// TwinCAT 3 PLC project mobject_nci
// Title: mobject-nci
// Company: mobject-io-ext
// Author: mobject dev team
// ProjectVersion: 0.0.1
// ProgramVersion: 3.1.4023.0
// libraries:
//   mobject-core, * (mobject.io)
//   mobject-motion, * (mobject-io-ext)
//   Tc2_NCI, * (Beckhoff Automation GmbH)
//   Tc2_PlcInterpolation, * (Beckhoff Automation GmbH)
//   Tc3_Module, * (Beckhoff Automation GmbH)
// project tree:
//   Lib/Feeder/ Feeder.TcPOU, I_Feeder.TcIO
//   Lib/NC-I/ ChannelType.TcDUT, I_Nci.TcIO, Nci.TcPOU, NciAxis.TcDUT, NciPlc.TcDUT
//   Lib/NC-I/Commands/ AddAxisToGroupCommand.TcPOU, BuildXYZGroupCommand.TcPOU, I_NciCommand.TcIO, NciCommand.TcPOU, ReleaseAxisCommand.TcPOU, ResetGroupCommand.TcPOU
//   Lib/Table/Enums/ FeedrateInterpolation.TcDUT, StandardPlane.TcDUT, TangentialFollowingBehaviour.TcDUT, VertexSmoothingBlendingType.TcDUT, VertexSmoothingSubType.TcDUT
//   Lib/Table/ I_Table.TcIO, Table.TcPOU

// ---- Lib/NC-I/ChannelType.TcDUT
{attribute 'qualified_only'}
{attribute 'strict'}
TYPE ChannelType :
(
	NONE := Tc2_PlcInterpolation.E_ItpChannelType.ItpChannelTypeNone,
	INTERPRETER := Tc2_PlcInterpolation.E_ItpChannelType.ItpChannelTypeInterpreter,
	KINEMATIC := Tc2_PlcInterpolation.E_ItpChannelType.ItpChannelTypeKinematic,
	INVALID_ITF_VERSION := Tc2_PlcInterpolation.E_ItpChannelType.ItpChannelType_InvalidItfVer
) INT;
END_TYPE

// ---- Lib/NC-I/NciAxis.TcDUT
{attribute 'qualified_only'}
{attribute 'strict'}
TYPE NciAxis :
(
	NONE := Tc2_PlcInterpolation.E_NciAxesInGroup.NoneAxis,
	X_AXIS := Tc2_PlcInterpolation.E_NciAxesInGroup.XAxis,
	Y_AXIS := Tc2_PlcInterpolation.E_NciAxesInGroup.YAxis,
	Z_AXIS := Tc2_PlcInterpolation.E_NciAxesInGroup.ZAxis,
	Q1_AXIS := Tc2_PlcInterpolation.E_NciAxesInGroup.Q1Axis,
	Q2_AXIS := Tc2_PlcInterpolation.E_NciAxesInGroup.Q2Axis,
	Q3_AXIS := Tc2_PlcInterpolation.E_NciAxesInGroup.Q3Axis,
	Q4_AXIS := Tc2_PlcInterpolation.E_NciAxesInGroup.Q4Axis,
	Q5_AXIS := Tc2_PlcInterpolation.E_NciAxesInGroup.Q5Axis
) INT;
END_TYPE

// ---- Lib/NC-I/NciPlc.TcDUT
TYPE NciPlc :
STRUCT
	nciToPlc AT %I* : NcToPlc_NciChannel_Ref;
	plcToNci AT %Q* : PlcToNc_NciChannel_Ref;
END_STRUCT
END_TYPE

// ---- Lib/Table/Enums/FeedrateInterpolation.TcDUT
{attribute 'qualified_only'}
{attribute 'strict'}
TYPE FeedrateInterpolation :
(
	CONST := Tc2_PlcInterpolation.E_NciFeedRateIpol.E_NciFeedrateIpolConstant,
    LINEAR := Tc2_PlcInterpolation.E_NciFeedRateIpol.E_NciFeedrateIpolLinear
) UINT;
END_TYPE

// ---- Lib/Table/Enums/StandardPlane.TcDUT
{attribute 'qualified_only'}
{attribute 'strict'}
TYPE StandardPlane :
(
	XY := Tc2_PlcInterpolation.E_NciGeoPlane.E_NciGeoPlaneXY,
	ZX := Tc2_PlcInterpolation.E_NciGeoPlane.E_NciGeoPlaneZX,
	YZ := Tc2_PlcInterpolation.E_NciGeoPlane.E_NciGeoPlaneYZ
) INT;
END_TYPE

// ---- Lib/Table/Enums/TangentialFollowingBehaviour.TcDUT
{attribute 'qualified_only'}
{attribute 'strict'}
TYPE TangentialFollowingBehaviour :
(
	IGNORE_ALL := Tc2_PlcInterpolation.E_TangentialFollowingBehavior.E_TfIngoreAll, // ignore critical angle
	ERROR_ON_EXCEEDING_CRITICAL_ANGLE := Tc2_PlcInterpolation.E_TangentialFollowingBehavior.E_TfErrorOnCritical1 // if angle becomes bigger than critical angle 1 ==> error
) INT;
END_TYPE

// ---- Lib/Table/Enums/VertexSmoothingBlendingType.TcDUT
{attribute 'qualified_only'}
{attribute 'strict'}
TYPE VertexSmoothingBlendingType :
(
	NONE := 0, // Probably should check this is correct!
	PARABOLIC := 2,
	BI_QUADRATIC := 3,
	BEZIER_3RD_ORDER := 4,
	BEZIER_5TH_ORDER := 5
) UDINT;
END_TYPE

// ---- Lib/Table/Enums/VertexSmoothingSubType.TcDUT
{attribute 'qualified_only'}
{attribute 'strict'}
TYPE VertexSmoothingSubType :
(
	NONE := 0, // Probably should check this is correct!
	CONSTANT_TOLERANCE_RADIUS := 1,
	DISTANCE_BETWEEN_INTERSETION_AND_VERTEX := 2,
	ADAPTIVE_TOLERANCE_RADIUS := 3
) UDINT;
END_TYPE

// ---- Lib/Feeder/I_Feeder.TcIO
INTERFACE I_Feeder EXTENDS __System.IQueryInterface

PROPERTY ChannelDone : BOOL
GET
END_GET
END_PROPERTY

METHOD FeedTable
VAR_INPUT
	table : I_Table;
	feedback : REFERENCE TO I_CommandFeedback;
END_VAR
END_METHOD

PROPERTY LogFeederEntries : BOOL
GET
END_GET
SET
END_SET
END_PROPERTY

METHOD Reset
VAR_INPUT
	feedback : REFERENCE TO I_CommandFeedback;
END_VAR
END_METHOD

END_INTERFACE

// ---- Lib/NC-I/Commands/I_NciCommand.TcIO
INTERFACE I_NciCommand EXTENDS I_Command

END_INTERFACE

// ---- Lib/NC-I/I_Nci.TcIO
INTERFACE I_Nci EXTENDS __System.IQueryInterface

PROPERTY _InternalNciPlcRef : REFERENCE TO NciPlc
GET
END_GET
END_PROPERTY

METHOD AddAxisToGroup
VAR_INPUT
	axis : I_Axis;
	index : UDINT;
	timeout : TIME;
	feedback : REFERENCE TO I_CommandFeedback;
END_VAR
END_METHOD

PROPERTY BlockNumber : UDINT
GET
END_GET
END_PROPERTY

METHOD BuildXYGroup
VAR_INPUT
	xAxis : I_Axis;
	yAxis : I_Axis;
	timeout : TIME;
	feedback : REFERENCE TO I_CommandFeedback;
END_VAR
END_METHOD

METHOD BuildXYZGroup
VAR_INPUT
	xAxis : I_Axis;
	yAxis : I_Axis;
	zAxis : I_Axis;
	timeout : TIME;
	feedback : REFERENCE TO I_CommandFeedback;
END_VAR
END_METHOD

PROPERTY ChannelId : UINT
GET
END_GET
END_PROPERTY

PROPERTY ChannelType : ChannelType
GET
END_GET
END_PROPERTY

PROPERTY ErrorId : UDINT
GET
END_GET
END_PROPERTY

METHOD GetGroupAxisIds : DWORD
VAR_IN_OUT
	axisIds : ARRAY[1..8] OF DWORD;
END_VAR
END_METHOD

METHOD GetOverride : LREAL
END_METHOD

PROPERTY GroupId : UDINT
GET
END_GET
END_PROPERTY

PROPERTY HandshakeableMFunction : INT
GET
END_GET
END_PROPERTY

PROPERTY HasError : BOOL
GET
END_GET
END_PROPERTY

PROPERTY HParam : DINT
GET
END_GET
END_PROPERTY

PROPERTY InterpreterState : UDINT
GET
END_GET
END_PROPERTY

PROPERTY IsEstop : BOOL
GET
END_GET
END_PROPERTY

METHOD IsFastMFunctionPresent : BOOL
VAR_INPUT
	functionNumber : INT;
END_VAR
END_METHOD

METHOD IsHandshakeableMFunctionPresent : BOOL
END_METHOD

METHOD ReadCyclicLRealParameter : LREAL
VAR_INPUT
	parameterNumber : UINT(1..4);
END_VAR
END_METHOD

METHOD ReadCyclicUdintParameter : UDINT
VAR_INPUT
	parameterNumber : UINT(1..4);
END_VAR
END_METHOD

METHOD ReleaseAxis
VAR_INPUT
	axis : I_Axis;
	timeout : TIME;
	feedback : REFERENCE TO I_CommandFeedback;
END_VAR
END_METHOD

METHOD ResetGroup
VAR_INPUT
	timeout : TIME;
	feedback : REFERENCE TO I_CommandFeedback;
END_VAR
END_METHOD

METHOD SetOverride : BOOL
VAR_INPUT
	value : LREAL;
END_VAR
END_METHOD

PROPERTY SetPathVelocity : LREAL
GET
END_GET
END_PROPERTY

PROPERTY SParam : UINT
GET
END_GET
END_PROPERTY

PROPERTY TParam : UINT
GET
END_GET
END_PROPERTY

END_INTERFACE

// ---- Lib/Table/I_Table.TcIO
INTERFACE I_Table EXTENDS __System.IQueryInterface

PROPERTY INTERNAL _InternalTable : REFERENCE TO ST_NciFeedGroupTable
GET
END_GET
END_PROPERTY

METHOD AddAxisDynamics : BOOL
VAR_INPUT
	displayIndex : UDINT;
    axis : I_Axis;
    acceleration : LREAL(0.000001-99999999);
    deceleration : LREAL(0.000001-99999999);
    jerk: LREAL(0.000001-99999999);
END_VAR
END_METHOD

METHOD AddBaseFrame : BOOL
VAR_INPUT
    displayIndex : UDINT;
    shiftX : LREAL;
    shiftY : LREAL;
    shiftZ : LREAL;
    rotationX : LREAL;
    rotationY : LREAL;
    rotationZ : LREAL;
    shiftQ1 : LREAL;
    shiftQ2 : LREAL;
    shiftQ3 : LREAL;
    shiftQ4 : LREAL;
    shiftQ5 : LREAL;
END_VAR
END_METHOD

METHOD AddBaseFrame3D : BOOL
VAR_INPUT
    displayIndex : UDINT;
    shiftX : LREAL;
    shiftY : LREAL;
    shiftZ : LREAL;
    rotationX : LREAL;
    rotationY : LREAL;
    rotationZ : LREAL;
END_VAR
END_METHOD

METHOD AddBezier3rdOrder : BOOL
VAR_INPUT
	displayIndex : UDINT;
    controlPoint1X : LREAL;
    controlPoint1Y : LREAL;
    controlPoint1Z : LREAL;
    controlPoint2X : LREAL;
    controlPoint2Y : LREAL;
    controlPoint2Z : LREAL;
	endPositionX : LREAL;
	endPositionY : LREAL;
	endPositionZ : LREAL;
	endPositionQ1 : LREAL;
	endPositionQ2 : LREAL;
	endPositionQ3 : LREAL;
	endPositionQ4 : LREAL;
	endPositionQ5 : LREAL;
	velocity : LREAL(0.000001-99999999);
	accurateStop : BOOL; // velocity at end == 0
END_VAR
END_METHOD

METHOD AddBezier3rdOrder3D : BOOL
VAR_INPUT
	displayIndex : UDINT;
    controlPoint1X : LREAL;
    controlPoint1Y : LREAL;
    controlPoint1Z : LREAL;
    controlPoint2X : LREAL;
    controlPoint2Y : LREAL;
    controlPoint2Z : LREAL;
	endPositionX : LREAL;
	endPositionY : LREAL;
	endPositionZ : LREAL;
	velocity : LREAL(0.000001-99999999);
	accurateStop : BOOL; // velocity at end == 0
END_VAR
END_METHOD

METHOD AddBezier5thOrder : BOOL
VAR_INPUT
	displayIndex : UDINT;
    controlPoint1X : LREAL;
    controlPoint1Y : LREAL;
    controlPoint1Z : LREAL;
    controlPoint2X : LREAL;
    controlPoint2Y : LREAL;
    controlPoint2Z : LREAL;
    controlPoint3X : LREAL;
    controlPoint3Y : LREAL;
    controlPoint3Z : LREAL;
    controlPoint4X : LREAL;
    controlPoint4Y : LREAL;
    controlPoint4Z : LREAL;
	endPositionX : LREAL;
	endPositionY : LREAL;
	endPositionZ : LREAL;
	endPositionQ1 : LREAL;
	endPositionQ2 : LREAL;
	endPositionQ3 : LREAL;
	endPositionQ4 : LREAL;
	endPositionQ5 : LREAL;
	velocity : LREAL(0.000001-99999999);
	accurateStop : BOOL; // velocity at end == 0
END_VAR
END_METHOD

METHOD AddBezier5thOrder3D : BOOL
VAR_INPUT
	displayIndex : UDINT;
    controlPoint1X : LREAL;
    controlPoint1Y : LREAL;
    controlPoint1Z : LREAL;
    controlPoint2X : LREAL;
    controlPoint2Y : LREAL;
    controlPoint2Z : LREAL;
    controlPoint3X : LREAL;
    controlPoint3Y : LREAL;
    controlPoint3Z : LREAL;
    controlPoint4X : LREAL;
    controlPoint4Y : LREAL;
    controlPoint4Z : LREAL;
	endPositionX : LREAL;
	endPositionY : LREAL;
	endPositionZ : LREAL;
	velocity : LREAL(0.000001-99999999);
	accurateStop : BOOL; // velocity at end == 0
END_VAR
END_METHOD

METHOD AddCircleCIP : BOOL
VAR_INPUT
	displayIndex : UDINT;
	endPositionX : LREAL;
	endPositionY : LREAL;
	endPositionZ : LREAL;
	arcPointX : LREAL;
	arcPointY : LREAL;
	arcPointZ : LREAL;
	endPositionQ1 : LREAL;
	endPositionQ2 : LREAL;
	endPositionQ3 : LREAL;
	endPositionQ4 : LREAL;
	endPositionQ5 : LREAL;
	velocity : LREAL(0.000001-99999999);
	accurateStop : BOOL; // velocity at end == 0
END_VAR
END_METHOD

METHOD AddCircleCIP3D : BOOL
VAR_INPUT
	displayIndex : UDINT;
	endPositionX : LREAL;
	endPositionY : LREAL;
	endPositionZ : LREAL;
	arcPointX : LREAL;
	arcPointY : LREAL;
	arcPointZ : LREAL;
	velocity : LREAL(0.000001-99999999);
	accurateStop : BOOL; // velocity at end == 0
END_VAR
END_METHOD

METHOD AddCircleOnPlane : BOOL
VAR_INPUT
	displayIndex : UDINT;
	endPositionX : LREAL;
	endPositionY : LREAL;
	endPositionZ : LREAL;
	centerX : LREAL;
	centerY : LREAL;
	centerZ : LREAL;
	endPositionQ1 : LREAL;
	endPositionQ2 : LREAL;
	endPositionQ3 : LREAL;
	endPositionQ4 : LREAL;
	endPositionQ5 : LREAL;
	plane : StandardPlane := StandardPlane.XY;
	clockwise : BOOL;
	velocity : LREAL(0.000001-99999999);
	accurateStop : BOOL; // velocity at end == 0
END_VAR
END_METHOD

METHOD AddCircleOnPlane3D : BOOL
VAR_INPUT
	displayIndex : UDINT;
	endPositionX : LREAL;
	endPositionY : LREAL;
	endPositionZ : LREAL;
	centerX : LREAL;
	centerY : LREAL;
	centerZ : LREAL;
	plane : StandardPlane := StandardPlane.XY;
	clockwise : BOOL;
	velocity : LREAL(0.000001-99999999);
	accurateStop : BOOL; // velocity at end == 0
END_VAR
END_METHOD

METHOD AddDwellTime : BOOL
VAR_INPUT
	displayIndex : UDINT;
    dwellTime : LREAL(0.000001-99999999); // seconds
END_VAR
END_METHOD

METHOD AddFeedrateInterpolation : BOOL
VAR_INPUT
	displayIndex : UDINT;
	interpolationType : FeedrateInterpolation;
END_VAR
END_METHOD

METHOD AddLine : BOOL
VAR_INPUT
    displayIndex: UDINT;
    endPositionX: LREAL;
    endPositionY: LREAL;
    endPositionZ: LREAL;
    endPositionQ1: LREAL;
    endPositionQ2: LREAL;
    endPositionQ3: LREAL;
    endPositionQ4: LREAL;
    endPositionQ5: LREAL;
    velocity: LREAL(0.000001-99999999);
    rapidTraverse: BOOL;
    accurateStop: BOOL; // velocity at end == 0
END_VAR
END_METHOD

METHOD AddLine3D : BOOL
VAR_INPUT
    displayIndex: UDINT;
    endPositionX: LREAL;
    endPositionY: LREAL;
    endPositionZ: LREAL;
    velocity: LREAL(0.000001-99999999);
    rapidTraverse: BOOL;
    accurateStop: BOOL; // velocity at end == 0
END_VAR
END_METHOD

METHOD AddMFunctionWithHandshake : BOOL
VAR_INPUT
	displayIndex : UDINT;
    functionNumber : INT(0..159);
END_VAR
END_METHOD

METHOD AddPathDynamics : BOOL
VAR_INPUT
    displayIndex : UDINT;
    acceleration : LREAL(0.000001-99999999);
    deceleration : LREAL(0.000001-99999999);
    jerk : LREAL(0.000001-99999999);
END_VAR
END_METHOD

METHOD AddStart : BOOL
VAR_INPUT
	x : LREAL;
	y : LREAL;
	z : LREAL;
	q1 : LREAL;
	q2 : LREAL;
	q3 : LREAL;
	q4 : LREAL;
	q5 : LREAL;
END_VAR
END_METHOD

METHOD AddStart3D : BOOL
VAR_INPUT
	x : LREAL;
	y : LREAL;
	z : LREAL;
END_VAR
END_METHOD

METHOD DisableTangentialFollowing : BOOL
END_METHOD

METHOD DisableVertexSmoothing : BOOL
VAR_INPUT
	displayIndex : UDINT;
END_VAR
END_METHOD

METHOD EnableTangentialFollowing : BOOL
VAR_INPUT
    tangentialAxis : NciAxis; // axis used for tangential following
    pathAxis1 : NciAxis; // describing the plane e.g. x
    pathAxis2 : NciAxis; // e.g. y ==> g17, xy plane
    offset : LREAL; // geo tangent is 0 degree, counting is mathmatical positive
	criticalAngle : LREAL(0.000001-90);
    behaviour : TangentialFollowingBehaviour;
END_VAR
END_METHOD

METHOD EnableVertexSmoothing : BOOL
VAR_INPUT
	displayIndex : UDINT;
	blendType : VertexSmoothingBlendingType;
	subType : VertexSmoothingSubType; 
	radius : LREAL(0.000001-99999999);
END_VAR
END_METHOD

METHOD End : BOOL
END_METHOD

PROPERTY ErrorId : UDINT
GET
END_GET
END_PROPERTY

PROPERTY FilledRows : INT
GET
END_GET
END_PROPERTY

PROPERTY HasError : BOOL
GET
END_GET
END_PROPERTY

METHOD ResetAll : BOOL
END_METHOD

METHOD ResetTable : BOOL
END_METHOD

END_INTERFACE

// ---- Lib/Feeder/Feeder.TcPOU
{attribute 'linkalways'} 
{attribute 'no_explicit_call' := 'This FB is a CLASS and must be accessed using methods or properties'}
FUNCTION_BLOCK Feeder EXTENDS CyclicInstance IMPLEMENTS I_Feeder
VAR
	_nci : I_Nci;
	_fb : FB_NciFeedTable;
	_table : ST_NciFeedGroupTable;
	_execute : BOOL;
	_reset : BOOL;
	_feedDone : BOOL;
	_channelDone : BOOL;
	_feedBusy : BOOL;
	_resetBusy : BOOL;
	_error : BOOL;
	_errorId : UDINT;
	
	state : (IDLE, RESETTING, FEEDING, DONE, ERROR);
	command : (NONE, RESET, FEED);
	
	commandFeedback : I_CommandFeedbackReadWrite;
	commandHasCompleted : BOOL;
	disposeOnceComplete : BOOL;
END_VAR

(*
	Beckhoff have put multiple functions into this function block that would
	normally be a few different function blocks. As such we emulate the
	I_Command behaviour internally as sharing a single function block across
	command instances seems a bit iffy.
*)

PROPERTY ChannelDone : BOOL
GET
ChannelDone := _fb.bChannelDone;
END_GET
END_PROPERTY

METHOD ClearFeedback
commandFeedback.Release();
commandFeedback := 0;
END_METHOD

METHOD CompleteTheCommand
ClearFeedback();

IF disposeOnceComplete THEN
	// DisposeCommand();
END_IF

// OnExecuteComplete();

commandHasCompleted := TRUE;
END_METHOD

METHOD  CyclicCall
CASE state OF
	IDLE:
		_fb(
			bExecute := FALSE,
			bReset := FALSE,
			stNciToPlc := _nci._InternalNciPlcRef.nciToPlc,
			stFeedGroupTable := _table,
		);
		
		CASE command OF
			RESET:
				state := RESETTING;
				command := NONE;
				commandFeedback.SetBusy();
			FEED:
				state := FEEDING;
				command := NONE;
				commandFeedback.SetBusy();
		END_CASE

	RESETTING:
		_fb(
			bExecute := FALSE,
			bReset := TRUE,
			stNciToPlc := _nci._InternalNciPlcRef.nciToPlc,
			stFeedGroupTable := _table,
		);
		
		IF NOT _fb.bResetBusy THEN		
			IF _fb.bError THEN
				state := ERROR;
			ELSE
				state := DONE;
			END_IF
		END_IF

	FEEDING:
		_fb(
			bExecute := TRUE,
			bReset := FALSE,
			stNciToPlc := _nci._InternalNciPlcRef.nciToPlc,
			stFeedGroupTable := _table,
		);
		
		IF NOT _fb.bFeedBusy THEN
			IF _fb.bError THEN
				state := ERROR;
			ELSIF _fb.bFeedingDone THEN
				state := DONE;
			END_IF
		END_IF
	
	DONE:
		IF commandFeedback <> 0 THEN
			commandFeedback.SetDone();
		END_IF
		state := IDLE;		
	ERROR:
		IF commandFeedback <> 0 THEN
			commandFeedback.SetError(_fb.nErrorId);
		END_IF
		state := IDLE;
ELSE
	state := IDLE;
END_CASE
END_METHOD

METHOD FB_init : BOOL
VAR_INPUT
	bInitRetains : BOOL; // if TRUE, the retain variables are initialized (warm start / cold start)
	bInCopyCode : BOOL;  // if TRUE, the instance afterwards gets moved into the copy code (online change)
	nci : I_Nci;
END_VAR
IF nci <> 0 THEN
	_nci := nci;
END_IF
END_METHOD

METHOD FeedTable
VAR_INPUT
	table : I_Table;
	feedback : REFERENCE TO I_CommandFeedback;
END_VAR
IF NOT IsAlreadyExecuting() THEN
	_table := table._InternalTable;
	command := FEED;
	SetupFeedback(feedback);
END_IF
END_METHOD

METHOD PRIVATE HasCompleted : BOOL
IF commandFeedback = 0 THEN
	HasCompleted := commandHasCompleted;
	RETURN;
END_IF

HasCompleted := NOT commandFeedback.Busy;
END_METHOD

METHOD PRIVATE IsAlreadyExecuting : BOOL
IF commandFeedback = 0 THEN
	RETURN;
END_IF

IsAlreadyExecuting := commandFeedback.Busy;
END_METHOD

METHOD PRIVATE IsStillBusyExecuting : BOOL
IF commandFeedback = 0 THEN
	RETURN;
END_IF

IsStillBusyExecuting := commandFeedback.Busy AND NOT commandFeedback.Aborting;
END_METHOD

PROPERTY LogFeederEntries : BOOL
GET
LogFeederEntries := _fb.bLogFeederEntries;
END_GET
SET
_fb.bLogFeederEntries := LogFeederEntries;
END_SET
END_PROPERTY

METHOD Reset
VAR_INPUT
	feedback : REFERENCE TO I_CommandFeedback;
END_VAR
IF NOT IsAlreadyExecuting() THEN
	command := RESET;
	SetupFeedback(Feedback);
END_IF
END_METHOD

METHOD SetupFeedback : I_CommandFeedbackReadWrite
VAR_INPUT
	feedback : REFERENCE TO I_CommandFeedback;
END_VAR
VAR
	pFeedback : POINTER TO CommandFeedback;
END_VAR
IF feedback <> 0 THEN 
	feedback.Release();
END_IF

IF IsAlreadyExecuting() THEN

	IF __ISVALIDREF(feedback) THEN
		feedback := commandFeedback;
		feedback.AddReference();
	END_IF
	
	RETURN;
END_IF

IF commandFeedback <> 0 THEN 
	commandFeedback.Release();
END_IF

pFeedback := __NEW(CommandFeedback);
commandFeedback := pFeedback^;

IF __ISVALIDREF(feedback) THEN
	feedback := commandFeedback;
	feedback.AddReference();
END_IF
END_METHOD

END_FUNCTION_BLOCK

// ---- Lib/NC-I/Nci.TcPOU
{attribute 'linkalways'} 
{attribute 'no_explicit_call' := 'This FB is a CLASS and must be accessed using methods or properties'}
FUNCTION_BLOCK Nci EXTENDS CyclicInstance IMPLEMENTS I_Nci
VAR
	_nciPlc : NciPlc;
END_VAR

PROPERTY _InternalNciPlcRef : REFERENCE TO NciPlc
GET
_InternalNciPlcRef REF= _nciPlc;
END_GET
END_PROPERTY

METHOD AddAxisToGroup
VAR_INPUT
	axis : I_Axis;
	index : UDINT;
	timeout : TIME;
	feedback : REFERENCE TO I_CommandFeedback;
END_VAR
VAR_INST
	pCmd : POINTER TO AddAxisToGroupCommand;
END_VAR
VAR
	_axis : I_Axis;
	_index : UDINT;
	_timeout : TIME;
END_VAR
_axis := axis;
_index := index;
_timeout := timeout;

pCmd := __NEW(AddAxisToGroupCommand(
	nci := THIS^,
	axis := _axis,
	index := _index,
	timeout := _timeout
));

(*
This doesn't work hence the horrible hack with intermediate values

pCmd := __NEW(AddAxisToGroupCommand(
	nci := THIS^,
	axis := axis,
	index := index,
	timeout := timeout
));
*)

pCmd^.Execute(feedback).ThenRelease();
END_METHOD

PROPERTY BlockNumber : UDINT
GET
BlockNumber := ItpGetBlockNumber(THIS^._nciPlc.nciToPlc);
END_GET
END_PROPERTY

METHOD BuildXYGroup
VAR_INPUT
	xAxis : I_Axis;
	yAxis : I_Axis;
	timeout : TIME;
	feedback : REFERENCE TO I_CommandFeedback;
END_VAR
VAR
	null : I_Axis;
END_VAR
BuildXYZGroup(xAxis, yAxis, null, timeout, feedback);
END_METHOD

METHOD BuildXYZGroup
VAR_INPUT
	xAxis : I_Axis;
	yAxis : I_Axis;
	zAxis : I_Axis;
	timeout : TIME;
	feedback : REFERENCE TO I_CommandFeedback;
END_VAR
VAR_INST
	pCmd : POINTER TO BuildXYZGroupCommand;
END_VAR
VAR
	_xAxis : I_Axis;
	_yAxis : I_Axis;
	_zAxis : I_Axis;
	_timeout : TIME;
END_VAR
_xAxis := xAxis;
_yAxis := yAxis;
_zAxis := zAxis;
_timeout := timeout;

pCmd := __NEW(BuildXYZGroupCommand(
	nci := THIS^,
	xAxis := _xAxis,
	yAxis := _yAxis,
	zAxis := _zAxis,
	timeout := _timeout
));

(*
This doesn't work hence the horrible hack with intermediate values

pCmd := __NEW(BuildXYZGroupCommand(
	nci := THIS^,
	xAxis := xAxis,
	yAxis := yAxis,
	zAxis := zAxis,
	timeout := commandTimeout
));
*)

pCmd^.Execute(feedback).ThenRelease();
END_METHOD

PROPERTY ChannelId : UINT
GET
ChannelId := ItpGetChannelId(THIS^._nciPlc.nciToPlc);
END_GET
END_PROPERTY

PROPERTY ChannelType : ChannelType
GET
VAR
	inter : INT;
	pInter : POINTER TO ChannelType;
END_VAR
// Don't know how to do the type conversion with NCIChannelType being strict
inter := ItpGetChannelType(THIS^._nciPlc.nciToPlc);
pInter := ADR(inter);
ChannelType := pInter^;
END_GET
END_PROPERTY

METHOD  CyclicCall
END_METHOD

PROPERTY ErrorId : UDINT
GET
ErrorId := ItpGetError(THIS^._nciPlc.nciToPlc);
END_GET
END_PROPERTY

METHOD GetGroupAxisIds : DWORD
VAR_IN_OUT
	axisIds : ARRAY[1..8] OF DWORD;
END_VAR
GetGroupAxisIds := ItpGetGroupAxisIds(axisIds, THIS^._nciPlc.nciToPlc);
END_METHOD

METHOD GetOverride : LREAL
GetOverride := ItpGetOverridePercent(THIS^._nciPlc.plcToNci);
END_METHOD

PROPERTY GroupId : UDINT
GET
GroupId := ItpGetGroupId(THIS^._nciPlc.nciToPlc);
END_GET
END_PROPERTY

PROPERTY HandshakeableMFunction : INT
GET
HandshakeableMFunction := ItpGetHskMFunc(THIS^._nciPlc.nciToPlc);
END_GET
END_PROPERTY

PROPERTY HasError : BOOL
GET
HasError := ItpHasError(THIS^._nciPlc.nciToPlc);
END_GET
END_PROPERTY

PROPERTY HParam : DINT
GET
HParam := ItpGetHParam(THIS^._nciPlc.nciToPlc);
END_GET
END_PROPERTY

PROPERTY InterpreterState : UDINT
GET
InterpreterState := ItpGetStateInterpreter(THIS^._nciPlc.nciToPlc);
END_GET
END_PROPERTY

PROPERTY IsEstop : BOOL
GET
IsEstop := ItpIsEStopEx(THIS^._nciPlc.nciToPlc);
END_GET
END_PROPERTY

METHOD IsFastMFunctionPresent : BOOL
VAR_INPUT
	functionNumber : INT;
END_VAR
IsFastMFunctionPresent := ItpIsFastMFunc(functionNumber, THIS^._nciPlc.nciToPlc);
END_METHOD

METHOD IsHandshakeableMFunctionPresent : BOOL
IsHandshakeableMFunctionPresent := ItpIsHskMFunc(THIS^._nciPlc.nciToPlc);
END_METHOD

METHOD ReadCyclicLRealParameter : LREAL
VAR_INPUT
	parameterNumber : UINT(1..4);
END_VAR
CASE parameterNumber OF
	1: ReadCyclicLRealParameter := ItpReadCyclicLRealParam1(THIS^._nciPlc.nciToPlc);
	2: ReadCyclicLRealParameter := ItpReadCyclicLRealParam2(THIS^._nciPlc.nciToPlc);
	3: ReadCyclicLRealParameter := ItpReadCyclicLRealParam3(THIS^._nciPlc.nciToPlc);
	4: ReadCyclicLRealParameter := ItpReadCyclicLRealParam4(THIS^._nciPlc.nciToPlc);
END_CASE
END_METHOD

METHOD ReadCyclicUdintParameter : UDINT
VAR_INPUT
	parameterNumber : UINT(1..4);
END_VAR
CASE parameterNumber OF
	1: ReadCyclicUdintParameter := ItpReadCyclicUdintParam1(THIS^._nciPlc.nciToPlc);
	2: ReadCyclicUdintParameter := ItpReadCyclicUdintParam2(THIS^._nciPlc.nciToPlc);
	3: ReadCyclicUdintParameter := ItpReadCyclicUdintParam3(THIS^._nciPlc.nciToPlc);
	4: ReadCyclicUdintParameter := ItpReadCyclicUdintParam4(THIS^._nciPlc.nciToPlc);
END_CASE
END_METHOD

METHOD ReleaseAxis
VAR_INPUT
	axis : I_Axis;
	timeout : TIME;
	feedback : REFERENCE TO I_CommandFeedback;
END_VAR
VAR_INST
	pCmd : POINTER TO ReleaseAxisCommand;
END_VAR
VAR
	_axis : I_Axis;
	_timeout : TIME;
END_VAR
_axis := axis;
_timeout := timeout;

pCmd := __NEW(ReleaseAxisCommand(
	axis := _axis,
	timeout := _timeout
));

(*
This doesn't work hence the horrible hack with intermediate values

pCmd := __NEW(ReleaseAxisCommand(
	axis := axis,
	timeout := timeout
));
*)
pCmd^.Execute(feedback).ThenRelease();
END_METHOD

METHOD ResetGroup
VAR_INPUT
	timeout : TIME;
	feedback : REFERENCE TO I_CommandFeedback;
END_VAR
VAR_INST
	pCmd : POINTER TO ResetGroupCommand;
END_VAR
VAR
	_timeout : TIME;
END_VAR
_timeout := timeout;

pCmd := __NEW(ResetGroupCommand(
	nci := THIS^,
	timeout := _timeout
));

(*
This doesn't work hence the horrible hack with intermediate values

pCmd := __NEW(ResetGroupCommand(
	nci := THIS^,
	timeout := timeout
));
*)

pCmd^.Execute(feedback).ThenRelease();
END_METHOD

METHOD SetOverride : BOOL
VAR_INPUT
	value : LREAL;
END_VAR
SetOverride := ItpSetOverridePercent(value, THIS^._nciPlc.plcToNci);
END_METHOD

PROPERTY SetPathVelocity : LREAL
GET
SetPathVelocity := ItpGetSetPathVelocity(THIS^._nciPlc.nciToPlc);
END_GET
END_PROPERTY

PROPERTY SParam : UINT
GET
SParam := ItpGetSParam(THIS^._nciPlc.nciToPlc);
END_GET
END_PROPERTY

PROPERTY TParam : UINT
GET
TParam := ItpGetTParam(THIS^._nciPlc.nciToPlc);
END_GET
END_PROPERTY

END_FUNCTION_BLOCK

// ---- Lib/NC-I/Commands/AddAxisToGroupCommand.TcPOU
{attribute 'linkalways'} 
{attribute 'no_explicit_call' := 'This FB is a CLASS and must be accessed using methods or properties'}
{attribute 'enable_dynamic_creation'}
FUNCTION_BLOCK AddAxisToGroupCommand EXTENDS NciCommand
VAR
	_fb : CfgAddAxisToGroup;
	_groupId : UDINT;
	_axisId : UDINT;
	_index : UDINT;
	_timeout : TIME;
END_VAR

METHOD FB_init : BOOL
VAR_INPUT
	bInitRetains : BOOL; // if TRUE, the retain variables are initialized (warm start / cold start)
	bInCopyCode : BOOL;  // if TRUE, the instance afterwards gets moved into the copy code (online change)
	nci : I_Nci;
	axis : I_Axis;
	index : UDINT;
	timeout : TIME;
END_VAR
IF nci <> 0 THEN
	_groupId := nci.GroupId;
END_IF
IF axis <> 0 THEN
	_axisId := axis.AxisId;
END_IF
_index := index;
_timeout := timeout;
END_METHOD

METHOD PROTECTED  WhileBusy
VAR_INPUT
	CommandState : I_CommandBusyState;
END_VAR
_fb(
	bExecute := TRUE,
	nGroupId := _groupId,
	nAxisId := _axisId,
	nIndex := _index,
	tTimeOut := _timeout
);

IF _fb.bBusy THEN
	RETURN;
END_IF

IF _fb.bErr THEN
	CommandState.SetError(_fb.nErrId);
	_fb(bExecute := FALSE);
	RETURN;
END_IF

_fb(bExecute := FALSE);
CommandState.SetDone();
END_METHOD

END_FUNCTION_BLOCK

// ---- Lib/NC-I/Commands/NciCommand.TcPOU
{attribute 'linkalways'} 
{attribute 'no_explicit_call' := 'This FB is a CLASS and must be accessed using methods or properties'}
{attribute 'enable_dynamic_creation'}
FUNCTION_BLOCK ABSTRACT NciCommand EXTENDS Command IMPLEMENTS I_NciCommand

END_FUNCTION_BLOCK

// ---- Lib/NC-I/Commands/BuildXYZGroupCommand.TcPOU
{attribute 'linkalways'} 
{attribute 'no_explicit_call' := 'This FB is a CLASS and must be accessed using methods or properties'}
{attribute 'enable_dynamic_creation'}
FUNCTION_BLOCK BuildXYZGroupCommand EXTENDS NciCommand
VAR
	_fb : CfgBuild3DGroup;
	_groupId : UDINT;
	_xAxisId : UDINT;
	_yAxisId : UDINT;
	_zAxisId : UDINT;
	_timeout : TIME;
END_VAR

METHOD FB_init : BOOL
VAR_INPUT
	bInitRetains : BOOL; // if TRUE, the retain variables are initialized (warm start / cold start)
	bInCopyCode : BOOL;  // if TRUE, the instance afterwards gets moved into the copy code (online change)
	nci : I_Nci := 0;
	xAxis : I_Axis := 0;
	yAxis : I_Axis := 0;
	zAxis : I_Axis := 0;
	timeout : TIME;
END_VAR
_groupId := nci.GroupId;
IF xAxis <> 0 THEN
	_xAxisId := xAxis.AxisId;
END_IF
IF yAxis <> 0 THEN
	_yAxisId := yAxis.AxisId;
END_IF
IF zAxis <> 0 THEN
	_zAxisId := zAxis.AxisId;
END_IF
_timeout := timeout;
END_METHOD

METHOD PROTECTED  WhileBusy
VAR_INPUT
	CommandState : I_CommandBusyState;
END_VAR
_fb(
	bExecute := TRUE,
	nGroupId := _groupId,
	nXAxisId := _xAxisId,
	nYAxisId := _yAxisId,
	nZAxisId := _zAxisId,
	tTimeOut := _timeout,
);

IF _fb.bBusy THEN
	RETURN;
END_IF

IF _fb.bErr THEN
	CommandState.SetError(_fb.nErrId);
	_fb(bExecute := FALSE);
	RETURN;
END_IF

_fb(bExecute := FALSE);
CommandState.SetDone();
END_METHOD

END_FUNCTION_BLOCK

// ---- Lib/NC-I/Commands/ReleaseAxisCommand.TcPOU
{attribute 'linkalways'} 
{attribute 'no_explicit_call' := 'This FB is a CLASS and must be accessed using methods or properties'}
{attribute 'enable_dynamic_creation'}
FUNCTION_BLOCK ReleaseAxisCommand EXTENDS NciCommand
VAR
	_fb : CfgReconfigAxis;
	_axisId : UDINT;
	_timeout : TIME;
END_VAR

METHOD FB_init : BOOL
VAR_INPUT
	bInitRetains : BOOL; // if TRUE, the retain variables are initialized (warm start / cold start)
	bInCopyCode : BOOL;  // if TRUE, the instance afterwards gets moved into the copy code (online change)
	axis : I_Axis;
	timeout : TIME;
END_VAR
IF axis <> 0 THEN
	_axisId := axis.AxisId;
END_IF
_timeout := timeout;
END_METHOD

METHOD PROTECTED  WhileBusy
VAR_INPUT
	CommandState : I_CommandBusyState;
END_VAR
_fb(
	bExecute := TRUE,
	nAxisId := _axisId,
	tTimeOut := _timeout
);

IF _fb.bBusy THEN
	RETURN;
END_IF

IF _fb.bErr THEN
	CommandState.SetError(_fb.nErrId);
	_fb(bExecute := FALSE);
	RETURN;
END_IF

_fb(bExecute := FALSE);
CommandState.SetDone();
END_METHOD

END_FUNCTION_BLOCK

// ---- Lib/NC-I/Commands/ResetGroupCommand.TcPOU
{attribute 'linkalways'} 
{attribute 'no_explicit_call' := 'This FB is a CLASS and must be accessed using methods or properties'}
{attribute 'enable_dynamic_creation'}
FUNCTION_BLOCK ResetGroupCommand EXTENDS NciCommand
VAR
	_fb : CfgReconfigGroup;
	_groupId : UDINT;
	_timeout : TIME;
END_VAR

METHOD FB_init : BOOL
VAR_INPUT
	bInitRetains : BOOL; // if TRUE, the retain variables are initialized (warm start / cold start)
	bInCopyCode : BOOL;  // if TRUE, the instance afterwards gets moved into the copy code (online change)
	nci : I_Nci;
	timeout : TIME;
END_VAR
IF nci <> 0 THEN
	_groupId := nci.GroupId;
END_IF
_timeout := timeout;
END_METHOD

METHOD PROTECTED  WhileBusy
VAR_INPUT
	CommandState : I_CommandBusyState;
END_VAR
_fb(
	bExecute := TRUE,
	nGroupId := _groupId,
	tTimeOut := _timeout
);

IF _fb.bBusy THEN
	RETURN;
END_IF

IF _fb.bErr THEN
	CommandState.SetError(_fb.nErrId);
	_fb(bExecute := FALSE);
	RETURN;
END_IF

_fb(bExecute := FALSE);
CommandState.SetDone();
END_METHOD

END_FUNCTION_BLOCK

// ---- Lib/Table/Table.TcPOU
{attribute 'linkalways'} 
{attribute 'no_explicit_call' := 'This FB is a CLASS and must be accessed using methods or properties'}
{attribute 'enable_dynamic_creation'}
FUNCTION_BLOCK Table IMPLEMENTS I_Table
VAR
	_fb : FB_NciFeedTablePreparation;
	_table : ST_NciFeedGroupTable;
	
	_stopped : STRING;
	_errorId : UDINT;
	_filledRows : INT;
END_VAR

PROPERTY _InternalTable : REFERENCE TO Tc2_PlcInterpolation.ST_NciFeedGroupTable
GET
_InternalTable REF= _table;
END_GET
END_PROPERTY

METHOD AddAxisDynamics : BOOL
VAR_INPUT
	displayIndex : UDINT;
	axis : mobject_motion.I_Axis;
	acceleration : LREAL(0.000001-99999999);
	deceleration : LREAL(0.000001-99999999);
	jerk : LREAL(0.000001-99999999);
END_VAR
VAR
	entry : ST_NciAxisDynamics;
END_VAR
entry.nDisplayIndex := displayIndex;
entry.nAxis := axis.AxisId;
entry.fAcc := acceleration;
entry.fDec := deceleration;
entry.fJerk := jerk;

_fb(
	stFeedGroupTable := _table,
	pEntry := ADR(entry),
	nEntryType := Tc2_PlcInterpolation.E_NciEntryType.E_NciEntryTypeAxisDynamics,
	bResetTable := FALSE,
	bResetAll := FALSE,
	nFilledRows => _filledRows
);

AddAxisDynamics := _fb.bError;
END_METHOD

METHOD AddBaseFrame : BOOL
VAR_INPUT
	displayIndex : UDINT;
	shiftX : LREAL;
	shiftY : LREAL;
	shiftZ : LREAL;
	rotationX : LREAL;
	rotationY : LREAL;
	rotationZ : LREAL;
	shiftQ1 : LREAL;
	shiftQ2 : LREAL;
	shiftQ3 : LREAL;
	shiftQ4 : LREAL;
	shiftQ5 : LREAL;
END_VAR
VAR
	entry : ST_NciBaseFrame;
END_VAR
entry.nDisplayIndex := displayIndex;
entry.fShiftX := shiftX;
entry.fShiftY := shiftY;
entry.fShiftZ := shiftZ;
entry.fRotX := rotationX;
entry.fRotY := rotationY;
entry.fRotZ := rotationZ;
entry.fShiftQ1 := shiftQ1;
entry.fShiftQ2 := shiftQ2;
entry.fShiftQ3 := shiftQ3;
entry.fShiftQ4 := shiftQ4;
entry.fShiftQ5 := shiftQ5;

_fb(
	stFeedGroupTable := _table,
	pEntry := ADR(entry),
	nEntryType := Tc2_PlcInterpolation.E_NciEntryType.E_NciEntryTypeBaseFrame,
	bResetTable := FALSE,
	bResetAll := FALSE,
	nFilledRows => _filledRows
);

AddBaseFrame := _fb.bError;
END_METHOD

METHOD AddBaseFrame3D : BOOL
VAR_INPUT
	displayIndex : UDINT;
	shiftX : LREAL;
	shiftY : LREAL;
	shiftZ : LREAL;
	rotationX : LREAL;
	rotationY : LREAL;
	rotationZ : LREAL;
END_VAR
AddBaseFrame3D := AddBaseFrame(
	displayIndex,
	shiftX, shiftY, shiftZ,
	rotationX, rotationY, rotationZ,
	0, 0, 0, 0, 0
);
END_METHOD

METHOD AddBezier3rdOrder : BOOL
VAR_INPUT
	displayIndex : UDINT;
	controlPoint1X : LREAL;
	controlPoint1Y : LREAL;
	controlPoint1Z : LREAL;
	controlPoint2X : LREAL;
	controlPoint2Y : LREAL;
	controlPoint2Z : LREAL;
	endPositionX : LREAL;
	endPositionY : LREAL;
	endPositionZ : LREAL;
	endPositionQ1 : LREAL;
	endPositionQ2 : LREAL;
	endPositionQ3 : LREAL;
	endPositionQ4 : LREAL;
	endPositionQ5 : LREAL;
	velocity : LREAL(0.000001-99999999);
	accurateStop : BOOL; // velocity at end == 0
END_VAR
VAR
	entry : ST_NciGeoBezier3;
END_VAR
entry.nDisplayIndex := displayIndex;
entry.fControlPoint1X := controlPoint1X;
entry.fControlPoint1Y := controlPoint1Y;
entry.fControlPoint1Z := controlPoint1Z;
entry.fControlPoint2X := controlPoint2X;
entry.fControlPoint2Y := controlPoint2Y;
entry.fControlPoint2Z := controlPoint2Z;
entry.fEndPosX := endPositionX;
entry.fEndPosY := endPositionY;
entry.fEndPosZ := endPositionZ;
entry.fEndPosQ1 := endPositionQ1;
entry.fEndPosQ2 := endPositionQ2;
entry.fEndPosQ3 := endPositionQ3;
entry.fEndPosQ4 := endPositionQ4;
entry.fEndPosQ5 := endPositionQ5;
entry.fVelo := velocity;
entry.bAccurateStop := accurateStop;

_fb(
	stFeedGroupTable := _table,
	pEntry := ADR(entry),
	nEntryType := Tc2_PlcInterpolation.E_NciEntryType.E_NciEntryTypeGeoBezier3,
	bResetTable := FALSE,
	bResetAll := FALSE,
	nFilledRows => _filledRows
);

AddBezier3rdOrder := _fb.bError;
END_METHOD

METHOD AddBezier3rdOrder3D : BOOL
VAR_INPUT
	displayIndex : UDINT;
	controlPoint1X : LREAL;
	controlPoint1Y : LREAL;
	controlPoint1Z : LREAL;
	controlPoint2X : LREAL;
	controlPoint2Y : LREAL;
	controlPoint2Z : LREAL;
	endPositionX : LREAL;
	endPositionY : LREAL;
	endPositionZ : LREAL;
	velocity : LREAL(0.000001-99999999);
	accurateStop : BOOL; // velocity at end == 0
END_VAR
AddBezier3rdOrder3D := AddBezier3rdOrder(
	displayIndex,
	controlPoint1X, controlPoint1Y, controlPoint1Z,
	controlPoint2X, controlPoint2Y, controlPoint2Z,
	endPositionX, endPositionY, endPositionZ,
	0, 0, 0, 0, 0,
	velocity,
	accurateStop
);
END_METHOD

METHOD AddBezier5thOrder : BOOL
VAR_INPUT
	displayIndex : UDINT;
	controlPoint1X : LREAL;
	controlPoint1Y : LREAL;
	controlPoint1Z : LREAL;
	controlPoint2X : LREAL;
	controlPoint2Y : LREAL;
	controlPoint2Z : LREAL;
	controlPoint3X : LREAL;
	controlPoint3Y : LREAL;
	controlPoint3Z : LREAL;
	controlPoint4X : LREAL;
	controlPoint4Y : LREAL;
	controlPoint4Z : LREAL;
	endPositionX : LREAL;
	endPositionY : LREAL;
	endPositionZ : LREAL;
	endPositionQ1 : LREAL;
	endPositionQ2 : LREAL;
	endPositionQ3 : LREAL;
	endPositionQ4 : LREAL;
	endPositionQ5 : LREAL;
	velocity : LREAL(0.000001-99999999);
	accurateStop : BOOL; // velocity at end == 0
END_VAR
VAR
	entry : ST_NciGeoBezier5;
END_VAR
entry.nDisplayIndex := displayIndex;
entry.fControlPoint1X := controlPoint1X;
entry.fControlPoint1Y := controlPoint1Y;
entry.fControlPoint1Z := controlPoint1Z;
entry.fControlPoint2X := controlPoint2X;
entry.fControlPoint2Y := controlPoint2Y;
entry.fControlPoint2Z := controlPoint2Z;
entry.fControlPoint3X := controlPoint3X;
entry.fControlPoint3Y := controlPoint3Y;
entry.fControlPoint3Z := controlPoint3Z;
entry.fControlPoint4X := controlPoint4X;
entry.fControlPoint4Y := controlPoint4Y;
entry.fControlPoint4Z := controlPoint4Z;
entry.fEndPosX := endPositionX;
entry.fEndPosY := endPositionY;
entry.fEndPosZ := endPositionZ;
entry.fEndPosQ1 := endPositionQ1;
entry.fEndPosQ2 := endPositionQ2;
entry.fEndPosQ3 := endPositionQ3;
entry.fEndPosQ4 := endPositionQ4;
entry.fEndPosQ5 := endPositionQ5;
entry.fVelo := velocity;
entry.bAccurateStop := accurateStop;

_fb(
	stFeedGroupTable := _table,
	pEntry := ADR(entry),
	nEntryType := Tc2_PlcInterpolation.E_NciEntryType.E_NciEntryTypeGeoBezier5,
	bResetTable := FALSE,
	bResetAll := FALSE,
	nFilledRows => _filledRows
);

AddBezier5thOrder := _fb.bError;
END_METHOD

METHOD AddBezier5thOrder3D : BOOL
VAR_INPUT
	displayIndex : UDINT;
	controlPoint1X : LREAL;
	controlPoint1Y : LREAL;
	controlPoint1Z : LREAL;
	controlPoint2X : LREAL;
	controlPoint2Y : LREAL;
	controlPoint2Z : LREAL;
	controlPoint3X : LREAL;
	controlPoint3Y : LREAL;
	controlPoint3Z : LREAL;
	controlPoint4X : LREAL;
	controlPoint4Y : LREAL;
	controlPoint4Z : LREAL;
	endPositionX : LREAL;
	endPositionY : LREAL;
	endPositionZ : LREAL;
	velocity : LREAL(0.000001-99999999);
	accurateStop : BOOL; // velocity at end == 0
END_VAR
AddBezier5thOrder3D := AddBezier5thOrder(
	displayIndex,
	controlPoint1X, controlPoint1Y, controlPoint1Z,
	controlPoint2X, controlPoint2Y, controlPoint2Z,
	controlPoint3X, controlPoint3Y, controlPoint3Z,
	controlPoint4X, controlPoint4Y, controlPoint4Z,
	endPositionX, endPositionY, endPositionZ,
	0, 0, 0, 0, 0,
	velocity,
	accurateStop
);
END_METHOD

METHOD AddCircleCIP : BOOL
VAR_INPUT
	displayIndex : UDINT;
	endPositionX : LREAL;
	endPositionY : LREAL;
	endPositionZ : LREAL;
	arcPointX : LREAL;
	arcPointY : LREAL;
	arcPointZ : LREAL;
	endPositionQ1 : LREAL;
	endPositionQ2 : LREAL;
	endPositionQ3 : LREAL;
	endPositionQ4 : LREAL;
	endPositionQ5 : LREAL;
	velocity : LREAL(0.000001-99999999);
	accurateStop : BOOL; // velocity at end == 0
END_VAR
VAR
	entry : ST_NciGeoCircleCIP;
END_VAR
entry.nDisplayIndex := displayIndex;
entry.fEndPosX := endPositionX;
entry.fEndPosY := endPositionY;
entry.fEndPosZ := endPositionZ;
entry.fCIPPosX := arcPointX;
entry.fCIPPosY := arcPointY;
entry.fCIPPosZ := arcPointZ;
entry.fEndPosQ1 := endPositionQ1;
entry.fEndPosQ2 := endPositionQ2;
entry.fEndPosQ3 := endPositionQ3;
entry.fEndPosQ4 := endPositionQ4;
entry.fEndPosQ5 := endPositionQ5;
entry.fVelo := velocity;
entry.bAccurateStop := accurateStop;

_fb(
	stFeedGroupTable := _table,
	pEntry := ADR(entry),
	nEntryType := Tc2_PlcInterpolation.E_NciEntryType.E_NciEntryTypeGeoCircleCIP,
	bResetTable := FALSE,
	bResetAll := FALSE,
	nFilledRows => _filledRows
);

AddCircleCIP := _fb.bError;
END_METHOD

METHOD AddCircleCIP3D : BOOL
VAR_INPUT
	displayIndex : UDINT;
	endPositionX : LREAL;
	endPositionY : LREAL;
	endPositionZ : LREAL;
	arcPointX : LREAL;
	arcPointY : LREAL;
	arcPointZ : LREAL;
	velocity : LREAL(0.000001-99999999);
	accurateStop : BOOL; // velocity at end == 0
END_VAR
AddCircleCIP3D := AddCircleCIP(
	displayIndex,
	endPositionX, endPositionY, endPositionZ,
	arcPointX, arcPointY, arcPointZ,
	0, 0, 0, 0, 0,
	velocity,
	accurateStop
);
END_METHOD

METHOD AddCircleOnPlane : BOOL
VAR_INPUT
	displayIndex : UDINT;
	endPositionX : LREAL;
	endPositionY : LREAL;
	endPositionZ : LREAL;
	centerX : LREAL;
	centerY : LREAL;
	centerZ : LREAL;
	endPositionQ1 : LREAL;
	endPositionQ2 : LREAL;
	endPositionQ3 : LREAL;
	endPositionQ4 : LREAL;
	endPositionQ5 : LREAL;
	plane : StandardPlane := StandardPlane.XY;
	clockwise : BOOL;	
	velocity : LREAL(0.000001-99999999);
	accurateStop : BOOL; // velocity at end == 0
END_VAR
VAR
	entry: ST_NciGeoCirclePlane;
END_VAR
entry.nDisplayIndex := displayIndex;
entry.fEndPosX := endPositionX;
entry.fEndPosY := endPositionY;
entry.fEndPosZ := endPositionZ;
entry.fCenterX := centerX;
entry.fCenterY := centerY;
entry.fCenterZ := centerZ;
entry.fEndPosQ1 := endPositionQ1;
entry.fEndPosQ2 := endPositionQ2;
entry.fEndPosQ3 := endPositionQ3;
entry.fEndPosQ4 := endPositionQ4;
entry.fEndPosQ5 := endPositionQ5;
entry.nPlane := plane;
entry.bClockwise := clockwise;
entry.fVelo := velocity;
entry.bAccurateStop := accurateStop;

_fb(
	stFeedGroupTable := _table,
	pEntry := ADR(entry),
	nEntryType := Tc2_PlcInterpolation.E_NciEntryType.E_NciEntryTypeGeoCirclePlane,
	bResetTable := FALSE,
	bResetAll := FALSE,
	nFilledRows => _filledRows
);

AddCircleOnPlane := _fb.bError;
END_METHOD

METHOD AddCircleOnPlane3D : BOOL
VAR_INPUT
	displayIndex : UDINT;
	endPositionX : LREAL;
	endPositionY : LREAL;
	endPositionZ : LREAL;
	centerX : LREAL;
	centerY : LREAL;
	centerZ : LREAL;
	plane : StandardPlane := StandardPlane.XY;
	clockwise : BOOL;
	velocity : LREAL(0.000001-99999999);
	accurateStop : BOOL; // velocity at end == 0
END_VAR
AddCircleOnPlane3D := AddCircleOnPlane(
	displayIndex,
	endPositionX,
	endPositionY,
	endPositionZ,
	centerX ,
	centerY,
	centerZ,
	0, 0, 0, 0, 0,
	plane,
	clockwise,	
	velocity,
	accurateStop
);
END_METHOD

METHOD AddDwellTime : BOOL
VAR_INPUT
	displayIndex : UDINT;
	dwellTime : LREAL(0.000001-99999999); // seconds
END_VAR
VAR
	entry: ST_NciDwellTime;
END_VAR
entry.nDisplayIndex := displayIndex;
entry.fDwellTime := dwellTime;

_fb(
	stFeedGroupTable := _table,
	pEntry := ADR(entry),
	nEntryType := Tc2_PlcInterpolation.E_NciEntryType.E_NciEntryTypeDwellTime,
	bResetTable := FALSE,
	bResetAll := FALSE,
	nFilledRows => _filledRows
);

AddDwellTime := _fb.bError;
END_METHOD

METHOD AddFeedrateInterpolation : BOOL
VAR_INPUT
	displayIndex : UDINT;
	interpolationType : FeedrateInterpolation;
END_VAR
VAR
	entry : ST_NciFeedrateIpol;
END_VAR
entry.nDisplayIndex := displayIndex;
entry.eFeedrateIpol := interpolationType;

_fb(
	stFeedGroupTable := _table,
	pEntry := ADR(entry),
	nEntryType := Tc2_PlcInterpolation.E_NciEntryType.E_NciEntryTypeFeedrateIpol,
	bResetTable := FALSE,
	bResetAll := FALSE,
	nFilledRows => _filledRows
);

 AddFeedrateInterpolation:= _fb.bError;
END_METHOD

METHOD AddLine : BOOL
VAR_INPUT
	displayIndex : UDINT;
	endPositionX : LREAL;
	endPositionY : LREAL;
	endPositionZ : LREAL;
	endPositionQ1 : LREAL;
	endPositionQ2 : LREAL;
	endPositionQ3 : LREAL;
	endPositionQ4 : LREAL;
	endPositionQ5 : LREAL;
	velocity : LREAL(0.000001-99999999);
	rapidTraverse : BOOL;
	accurateStop : BOOL; // velocity at end == 0
END_VAR
VAR
	entry : ST_NciGeoLine;
END_VAR
entry.nDisplayIndex := displayIndex;
entry.fEndPosX := endPositionX;
entry.fEndPosY := endPositionY;
entry.fEndPosZ := endPositionZ;
entry.fEndPosQ1 := endPositionQ1;
entry.fEndPosQ2 := endPositionQ2;
entry.fEndPosQ3 := endPositionQ3;
entry.fEndPosQ4 := endPositionQ4;
entry.fEndPosQ5 := endPositionQ5;
entry.fVelo := velocity;
entry.bRapidTraverse := rapidTraverse;
entry.bAccurateStop := accurateStop;

_fb(
	stFeedGroupTable := _table,
	pEntry := ADR(entry),
	nEntryType := Tc2_PlcInterpolation.E_NciEntryType.E_NciEntryTypeGeoLine,
	bResetTable := FALSE,
	bResetAll := FALSE,
	nFilledRows => _filledRows
);

AddLine := _fb.bError;
END_METHOD

METHOD AddLine3D : BOOL
VAR_INPUT
	displayIndex : UDINT;
	endPositionX : LREAL;
	endPositionY : LREAL;
	endPositionZ : LREAL;
	velocity : LREAL(0.000001-99999999);
	rapidTraverse : BOOL;
	accurateStop : BOOL; // velocity at end == 0
END_VAR
AddLine3D := AddLine(
	displayIndex,
	endPositionX,
	endPositionY,
	endPositionZ,
	0, 0, 0, 0, 0,
	velocity,
	rapidTraverse,
	accurateStop
);
END_METHOD

METHOD AddMFunctionWithHandshake : BOOL
VAR_INPUT
	displayIndex : UDINT;
	functionNumber : INT(0..159);
END_VAR
VAR
	entry : ST_NciMFuncHsk;
END_VAR
entry.nDisplayIndex := displayIndex;
entry.nMFunc := functionNumber;

_fb(
	stFeedGroupTable := _table,
	pEntry := ADR(entry),
	nEntryType := Tc2_PlcInterpolation.E_NciEntryType.E_NciEntryTypeMFuncHsk,
	bResetTable := FALSE,
	bResetAll := FALSE,
	nFilledRows => _filledRows
);

 AddMFunctionWithHandshake := _fb.bError;
END_METHOD

METHOD AddPathDynamics : BOOL
VAR_INPUT
	displayIndex : UDINT;
	acceleration : LREAL(0.000001-99999999);
	deceleration : LREAL(0.000001-99999999);
	jerk : LREAL(0.000001-99999999);
END_VAR
VAR
	entry : ST_NciPathDynamics;
END_VAR
entry.nDisplayIndex := displayIndex;
entry.fAcc := acceleration;
entry.fDec := deceleration;
entry.fJerk := jerk;

_fb(
	stFeedGroupTable := _table,
	pEntry := ADR(entry),
	nEntryType := Tc2_PlcInterpolation.E_NciEntryType.E_NciEntryTypePathDynamics,
	bResetTable := FALSE,
	bResetAll := FALSE,
	nFilledRows => _filledRows
);

AddPathDynamics := _fb.bError;
END_METHOD

METHOD AddReference
END_METHOD

METHOD AddStart : BOOL
VAR_INPUT
	x : LREAL;
	y : LREAL;
	z : LREAL;
	q1 : LREAL;
	q2 : LREAL;
	q3 : LREAL;
	q4 : LREAL;
	q5 : LREAL;
END_VAR
VAR
	entry : ST_NciGeoStart;
END_VAR
entry.fPosX := x;
entry.fPosY := y;
entry.fPosZ := z;
entry.fPosQ1 := q1;
entry.fPosQ2 := q2;
entry.fPosQ3 := q3;
entry.fPosQ4 := q4;
entry.fPosQ5 := q5;

_fb(
	stFeedGroupTable := _table,
	pEntry := ADR(entry),
	nEntryType := Tc2_PlcInterpolation.E_NciEntryType.E_NciEntryTypeGeoStart,
	bResetTable := FALSE,
	bResetAll := FALSE,
	nFilledRows => _filledRows
);

AddStart := _fb.bError;
END_METHOD

METHOD AddStart3D : BOOL
VAR_INPUT
	x : LREAL;
	y : LREAL;
	z : LREAL;
END_VAR
AddStart3D := AddStart(x, y, z, 0, 0, 0, 0, 0);
END_METHOD

METHOD DisableTangentialFollowing : BOOL
VAR
	entry : ST_NciTangentialFollowingDesc;
END_VAR
entry.bTangOn := FALSE;

_fb(
	stFeedGroupTable := _table,
	pEntry := ADR(entry),
	nEntryType := Tc2_PlcInterpolation.E_NciEntryType.E_NciEntryTypeTfDesc,
	bResetTable := FALSE,
	bResetAll := FALSE,
	nFilledRows => _filledRows
);

DisableTangentialFollowing := _fb.bError;
END_METHOD

METHOD DisableVertexSmoothing : BOOL
VAR_INPUT
	displayIndex : UDINT;
END_VAR
DisableVertexSmoothing := EnableVertexSmoothing(
	displayIndex,
	VertexSmoothingBlendingType.NONE,
	VertexSmoothingSubType.NONE,
	0
);
END_METHOD

METHOD EnableTangentialFollowing : BOOL
VAR_INPUT
	tangentialAxis : NciAxis; // axis used for tangential following
	pathAxis1 : NciAxis; // describing the plane e.g. x
	pathAxis2 : NciAxis; // e.g. y ==> g17, xy plane
	offset : LREAL; // geo tangent is 0 degree, counting is mathmatical positive
	criticalAngle : LREAL(0.000001-90);
	behaviour : TangentialFollowingBehaviour;
END_VAR
VAR
	entry : ST_NciTangentialFollowingDesc;
END_VAR
entry.bTangOn := TRUE;
entry.nTangAxis := tangentialAxis;
entry.nPathAxis1 := pathAxis1;
entry.nPathAxis2 := pathAxis2;
entry.fOffset := offset;
entry.fCriticalAngle1 := criticalAngle;
entry.nTfBehavior := behaviour;

_fb(
	stFeedGroupTable := _table,
	pEntry := ADR(entry),
	nEntryType := Tc2_PlcInterpolation.E_NciEntryType.E_NciEntryTypeTfDesc,
	bResetTable := FALSE,
	bResetAll := FALSE,
	nFilledRows => _filledRows
);

EnableTangentialFollowing := _fb.bError;
END_METHOD

METHOD EnableVertexSmoothing : BOOL
VAR_INPUT
	displayIndex : UDINT;
	blendType : VertexSmoothingBlendingType;
	subType : VertexSmoothingSubType;
	radius : LREAL(0.000001-99999999);
END_VAR
VAR
	entry : ST_NciVertexSmoothing;
END_VAR
entry.nEntryType := Tc2_PlcInterpolation.E_NciEntryType.E_NciEntryTypeVertexSmoothing;
entry.nDisplayIndex := displayIndex;
entry.nType := blendType;
entry.nSubtype :=	subType;
entry.fRadius :=	radius;

_fb(
	stFeedGroupTable := _table,
	pEntry := ADR(entry),
	nEntryType := Tc2_PlcInterpolation.E_NciEntryType.E_NciEntryTypeVertexSmoothing,
	bResetTable := FALSE,
	bResetAll := FALSE,
	nFilledRows => _filledRows
);

EnableVertexSmoothing := _fb.bError;
END_METHOD

METHOD End : BOOL
VAR
	entry : ST_NciEndOfTables;
END_VAR
_fb(
	stFeedGroupTable := _table,
	pEntry := ADR(entry),
	nEntryType := Tc2_PlcInterpolation.E_NciEntryType.E_NciEntryTypeEndOfTables,
	bResetTable := FALSE,
	bResetAll := FALSE,
	nFilledRows => _filledRows
);

End := _fb.bError;
END_METHOD

PROPERTY ErrorId : UDINT
GET
ErrorId := _fb.nErrorId;
END_GET
END_PROPERTY

PROPERTY FilledRows : INT
GET
FilledRows := _filledRows;
END_GET
END_PROPERTY

PROPERTY HasError : BOOL
GET
HasError := _fb.bError;
END_GET
END_PROPERTY

METHOD ResetAll : BOOL
_fb(
	stFeedGroupTable := _table,
	bResetAll := TRUE
);

ResetAll := _fb.bError;
END_METHOD

METHOD ResetTable : BOOL
_fb(
	stFeedGroupTable := _table,
	bResetTable := TRUE
);

ResetTable := _fb.bError;
END_METHOD

END_FUNCTION_BLOCK
